// TIA Portal V20 export
TYPE "LER_typeMobileRFIDInterface"
// stored: Access Published
   STRUCT
      commands : "LER_typeMobileRFIDCommands";
      monitoring : "LER_typeMobileRFIDMonitoring";
      configuration : "LER_typeMobileRFIDConfiguration";
   END_STRUCT;
END_TYPE
